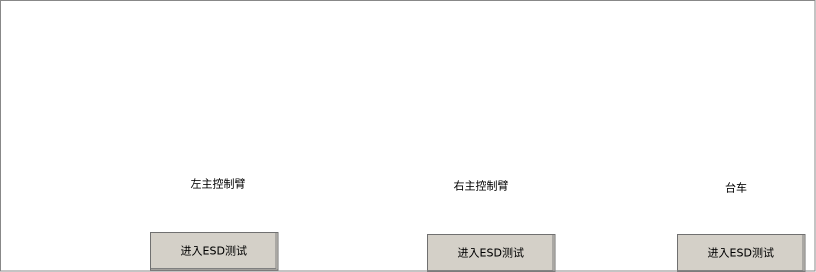
VISUALIZATION cycle_ESD  // 816x272
    Button (150,232 128x38), "进入ESD测试", colour toggle: g_cycleTest.m_enterESDTest[1]
        toggle g_cycleTest.m_enterESDTest[1]
    Label (138,153 160x62), "左主控制臂"
    Label (401,155 160x62), "右主控制臂"
    Label (656,157 160x62), "台车"
    Button (427,234 128x38), "进入ESD测试", colour toggle: g_cycleTest.m_enterESDTest[2]
        toggle g_cycleTest.m_enterESDTest[2]
    Button (677,234 128x38), "进入ESD测试", colour toggle: g_cycleTest.m_carEnterESDTest
        toggle g_cycleTest.m_carEnterESDTest
END_VISUALIZATION

(* stored: Version 1.1.0.1, ProductVersion 3.1.4024.11
   Visu cycle_ESD: Id {2444bc07-fcc1-417a-b488-668e29a68ad3} *)
